// TIA Portal project "PID_1" (V16)

(* hardware
DEVICE "S71500/ET200MP station_1"  S7-1500 station
   slot 0: "Rail_0"  Rack  6ES7 590-1***0-0AA0
   slot 1: "PLC_1"  CPU 1511C-1 PN  6ES7 511-1CK01-0AB0  V2.8
      slot 3: "CPU display_1"  6ES7591-1AA00-0AA0
      slot 32768: "PROFINET interface_1"  X1
         slot 32769: "Port_1"  X1 P1
         slot 32770: "Port_2"  X1 P2
      slot 34817: "Virtual CP interface port_1"  Virtual CP interface port  Virtual CP interface port
DEVICE "HMI_1"  KTP700 Basic PN
   slot 0: "HMI_1"  KTP700 Basic PN  6AV2 123-2GB03-0AX0  16.0.0.0
   slot 1: "HMI_RT_1"  KTP700 Basic PN  6AV2 123-2GB03-0AX0  16.0.0.0
   slot 5: "HMI_1.IE_CP_1"  PROFINET Interface  16.0.0.0
      slot 1: "PROFINET Interface_1"  PROFINET Interface
         slot 1: "Port_1"  Port
*)

// ===== PLC "PLC_1"  CPU 1511C-1 PN =====

VAR_GLOBAL   // PLC tag table "Default tag table"
   "Fill level Tank" AT %IW0 : Int;
   "Analog Output" AT %QW0 : Int;
   "Empty Tank" AT %I0.0 : Bool;
   "Fill In Tank" AT %I0.1 : Bool;
   "LED Indicator" AT %Q4.0 : Bool;
END_VAR

VAR_GLOBAL   // PLC tag table "Outputs"
   "Solenoid_on/off" AT %Q0.0 : Bool;
   "Heater_on/off" AT %Q0.1 : Bool;
   "Relay KF1_Pump mode" AT %Q0.2 : Bool;
   "Pump_on/off" AT %Q0.3 : Bool;
   "KF6_Proportional valve" AT %Q0.4 : Bool;
   "KF2_Fan" AT %Q0.5 : Bool;
   "Pump_P101" AT %QW96 : Int;
END_VAR

VAR_GLOBAL   // PLC tag table "Inputs"
   "Flow_Rate_Sensor" AT %I0.0 : Bool;
   "Float_switch_overflow" AT %I0.1 : Bool;   // S111
   "Float_switch_threshold" AT %I0.2 : Bool;   // S112
   "Low_Level_Capacitive_Sensor" AT %I0.3 : Bool;   // B114
   "High_Level_Capacitive_Sensor" AT %I0.4 : Bool;   // B113
   "Micro_switch_valve_closed" AT %I0.5 : Bool;
   "Micro_switch_valve_open" AT %I0.6 : Bool;
   "Ultrasonic_Sensor" AT %IW96 : Int;
END_VAR

VAR_GLOBAL   // PLC tag table "Factory tags"
   "FactoryIO_running" AT %I0.7 : Bool;
   "Ultrasonic_Sensor_factory" AT %ID30 : Real;
   "Fill valve" AT %QD30 : Real;
   "Discharge valve" AT %QD34 : Real;
   "SP" AT %QD38 : DInt;
   "Flow meter" AT %ID34 : Real;
   "setpoint" AT %ID38 : DInt;
   "PV" AT %QD42 : Real;
END_VAR

// folder: Sys_par

DATA_BLOCK "parameters"   // DB4
{ S7_Optimized_Access := 'TRUE' }
VERSION : 0.1
   VAR
      "Process Value" : Real;
      setpoint : Int := 0;
      flowrate : Real;
      ModeActivate : Bool;
      ManualEnable : Bool;
      ManualValue : Real := 80.0;
      Mode : Int;
      Reset : Bool;
   END_VAR
BEGIN
END_DATA_BLOCK

// folder: (top level)

FUNCTION "height_conversion" : Void   // FC3, LAD
{ S7_Optimized_Access := 'TRUE' }
VERSION : 0.1
   VAR_INPUT
      height_sensor : Real;
      height_setpoint : Int;
   END_VAR
   VAR_OUTPUT
      scaled_height : Real;
      scaled_setpoint : Real;
   END_VAR
   VAR_TEMP
      norm_height : Real;
      norm_setpoint : Real;
   END_VAR
BEGIN

REGION Network 1: Height Conversion
   // 1. Normalize the sensor output data between 0.0 and 1.0
   // 2. Scale the normalized data between minimum and maximum scale reading
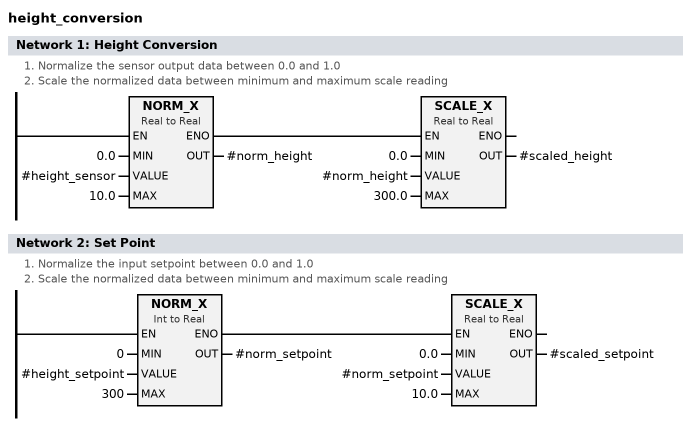
   RUNG wire#powerrail
      { S7_Templates := "[SrcType := Real, DestType := Real]" } Normalize(min := 0.0, value := #height_sensor, max := 10.0, out => #norm_height)
      { S7_Templates := "[SrcType := Real, DestType := Real]" } Scale(min := 0.0, value := #norm_height, max := 300.0, out => #scaled_height)
   END_RUNG
   // the same network as SCL:
   #norm_height := NORM_X(MIN := 0.0, VALUE := #height_sensor, MAX := 10.0);
   #scaled_height := SCALE_X(MIN := 0.0, VALUE := #norm_height, MAX := 300.0);
END_REGION

REGION Network 2: Set Point
   // 1. Normalize the input setpoint between 0.0 and 1.0
   // 2. Scale the normalized data between minimum and maximum scale reading
   RUNG wire#powerrail
      { S7_Templates := "[SrcType := Int, DestType := Real]" } Normalize(min := 0, value := #height_setpoint, max := 300, out => #norm_setpoint)
      { S7_Templates := "[SrcType := Real, DestType := Real]" } Scale(min := 0.0, value := #norm_setpoint, max := 10.0, out => #scaled_setpoint)
   END_RUNG
   // the same network as SCL:
   #norm_setpoint := NORM_X(MIN := 0, VALUE := #height_setpoint, MAX := 300);
   #scaled_setpoint := SCALE_X(MIN := 0.0, VALUE := #norm_setpoint, MAX := 10.0);
END_REGION
END_FUNCTION

FUNCTION "MHJ-PLC-Lab-Function-S71500" : Void   // FC9000, SCL
{ S7_Optimized_Access := 'TRUE' }
VERSION : 0.1
   VAR_TEMP
      Value : Byte;
      ForCounter : Int;
   END_VAR
   VAR CONSTANT
      Value_01_DW : DWord := 16#1223_5486;
      Value_02_DW : DWord := 16#A6C9_D1F5;
   END_VAR
BEGIN

   #Value:=PEEK(area := 16#82,
        dbNumber := 0,
        byteOffset := 511);
   #Value := #Value + 1;

   POKE(area := 16#82,
        dbNumber := 0,
        byteOffset := 511,
        value := #Value);

   POKE(area := 16#82,
        dbNumber := 0,
        byteOffset := 1016,
        value := #Value_01_DW);
   POKE(area := 16#82,
        dbNumber := 0,
        byteOffset := 1020,
        value := #Value_02_DW);

   FOR #ForCounter := 0 TO 63 DO
       #Value:=PEEK(area := 16#1,
            dbNumber := 0,
            byteOffset := #ForCounter);
       POKE(area := 16#81,
            dbNumber := 0,
            byteOffset := #ForCounter,
            value := #Value);
   END_FOR;
   #Value := PEEK(area := 16#1,
                  dbNumber := 0,
                  byteOffset := 512);
   POKE(area := 16#82,
        dbNumber := 0,
        byteOffset := 512,
        value := #Value);
END_FUNCTION

ORGANIZATION_BLOCK "Main"   // OB1, LAD, ProgramCycle
TITLE = "Main Program Sweep (Cycle)"
{ S7_Optimized_Access := 'TRUE' }
VERSION : 0.1
   VAR_INPUT
      Initial_Call : Bool;   // Initial call of this OB
      Remanence : Bool;   // =True, if remanent data are available
   END_VAR
BEGIN

REGION Network 1: Konnektierungsbaustein für PLC-Lab / Factory IO Function
   // Im Netzwerk 1 wird der Konnektierungsbaustein für PLC-Lab aufgerufen.
   // Dieser Aufruf darf nicht entfernt werden!
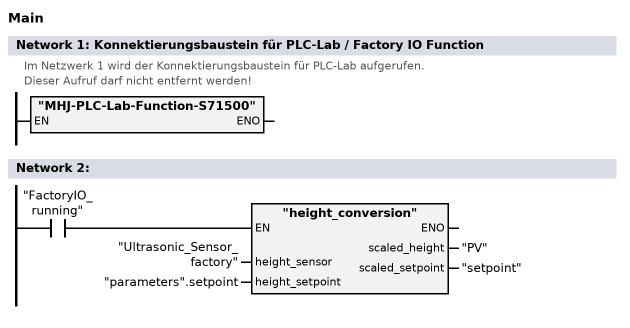
   RUNG wire#powerrail
      "MHJ-PLC-Lab-Function-S71500"()
   END_RUNG
   // the same network as SCL:
   "MHJ-PLC-Lab-Function-S71500"();
END_REGION

REGION Network 2
   RUNG wire#powerrail
      Contact( "FactoryIO_running" )
      "height_conversion"(height_sensor := "Ultrasonic_Sensor_factory", height_setpoint := "parameters".setpoint, scaled_height => "PV", scaled_setpoint => "setpoint")
   END_RUNG
   // the same network as SCL:
   IF "FactoryIO_running" THEN
       "height_conversion"(height_sensor := "Ultrasonic_Sensor_factory",
                           height_setpoint := "parameters".setpoint,
                           scaled_height => "PV",
                           scaled_setpoint => "setpoint");
   END_IF;
END_REGION
END_ORGANIZATION_BLOCK

ORGANIZATION_BLOCK "Cyclic interrupt PID"   // OB30, LAD, CyclicInterrupt
{ S7_Optimized_Access := 'TRUE' }
VERSION : 0.1
   VAR_INPUT
      Initial_Call : Bool;   // Initial call of this OB
      Event_Count : Int;   // Events discarded
   END_VAR
BEGIN

REGION Network 1
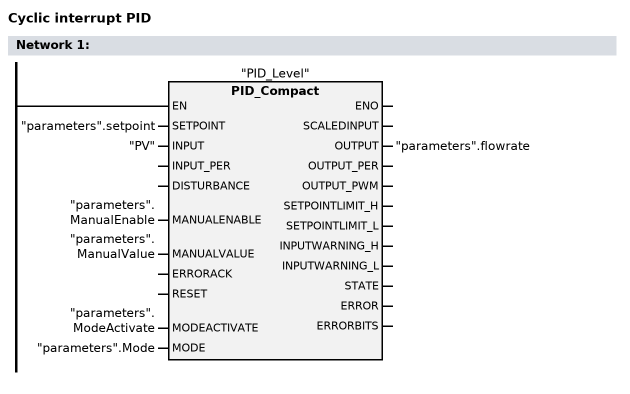
   "PID_Level"(Setpoint := "parameters".setpoint,   // PID_Compact
               Input := "PV",
               ManualEnable := "parameters".ManualEnable,
               ManualValue := "parameters".ManualValue,
               ModeActivate := "parameters".ModeActivate,
               Mode := "parameters".Mode,
               Output => "parameters".flowrate);
END_REGION
END_ORGANIZATION_BLOCK

(* ===== HMI "HMI_RT_1" =====
system functions are stored by id; their names below are inferred from use
connection "HMI_Connection_1": ETHERNET, SMART_S7_1200_OMS

HMI tags "Default tag table"
   "Tag_ScreenNumber" : UInt, internal
   "Float_switch_threshold" : Bool = PLC Float_switch_threshold AT %I0.2, 1 s
   "High_Level_Capacitive_Sensor" : Bool = PLC High_Level_Capacitive_Sensor AT %I0.4, 1 s
   "Low_Level_Capacitive_Sensor" : Bool = PLC Low_Level_Capacitive_Sensor AT %I0.3, 1 s
   "Float_switch_overflow" : Bool = PLC Float_switch_overflow AT %I0.1, 1 s
   "Micro_switch_valve_open" : Bool = PLC Micro_switch_valve_open AT %I0.6, 1 s
   "Micro_switch_valve_closed" : Bool = PLC Micro_switch_valve_closed AT %I0.5, 1 s
   "Relay KF1_Pump mode" : Bool = PLC "Relay KF1_Pump mode" AT %Q0.2, 1 s
   "KF6_Proportional valve" : Bool = PLC "KF6_Proportional valve" AT %Q0.4, 1 s
   "PV" : Real = PLC PV AT %QD42, 1 s
   "setpoint" : DInt = PLC setpoint AT %ID38, 1 s
   "PID_Compact_Level_CtrlParamsBackUp_Gain" : Real = PLC PID_Compact_Level.CtrlParamsBackUp.Gain, 1 s
   "PID_Compact_Level_CtrlParamsBackUp_Ti" : Real = PLC PID_Compact_Level.CtrlParamsBackUp.Ti, 1 s
   "PID_Compact_Level_CtrlParamsBackUp_Td" : Real = PLC PID_Compact_Level.CtrlParamsBackUp.Td, 1 s

HMI tags "Local Template"
   "_iScreenNumber" : Int, internal
   "_xState_Btn_Overview" : Bool, internal
   "_xState_Btn_Alarm" : Bool, internal
   "_xState_Btn_Recipe" : Bool, internal
   "_xState_Btn_Settings" : Bool, internal
   "_xState_Btn_Level_Overview" : Bool, internal
   "_xState_Btn_Level_Config" : Bool, internal
   "_xState_Btn_Alarm_Buffer" : Bool, internal

discrete alarms
   1: 'REFILL PROCESS 1 - PUMP- MOTOR CIRCUT BREAKER', class Errors
   2: 'REFILL PROCESS 1 - PUMP- LOCAL ISOLATOR FAULT', class Errors bit 0
   3: 'REFILL PROCESS 1 - PUMP- RUNNING FEEDBACK FAULT', class Errors bit 0
   4: 'REFILL PROCESS 1 - VALVE-NOT OPENING', class Errors bit 0
   5: 'SUPPLY-TANK-LOW LEVEL FAULT', class Errors bit 0
   6: 'SUPPLY-TANK-NOT OPENING FAULT', class Errors bit 0
   7: 'SUPPLY-TANK-HIGH LEVEL WARNING', class Warnings bit 0
   8: 'PROCESS-TANK-HIGH LEVEL ERROR', class Errors bit 0

graphic list "Graphic_Alarm_Reset": 0 'Graphic_49'; 1 'Graphic_50'

graphic list "Graphic_Return_Previous_Screen": 0..1 'Graphic_52'

graphic list "Graphic_Buffer_Screen": 0..1 'Graphic_54'

graphic list "GraphList_Btn_Template_Overview": 0 'Graphic_19'; 1 'Graphic_18'

graphic list "GraphList_Btn_Template_Alarm": 0 'Graphic_16'; 1 'Graphic_17'

graphic list "GraphList_Btn_Template_Recipe": 0 'Graphic_14'; 1 'Graphic_15'

graphic list "GraphList_Btn_Template_Settings": 0 'Graphic_13'; 1 'Graphic_12'

graphic list "GraphList_Pump": 0 'Graphic_27'; 1 'Graphic_26'

graphic list "GraphList_Proportional_Valve": 0 'Graphic_45'; 1 'Graphic_46'

screen "Overview" 800x480, template "Template"
   on GenerateScreen: SetBit("_xState_Btn_Overview")
   on ClearScreen: ResetBit("_xState_Btn_Overview")
   Button "Button_1" at 140,201 size 182x58; TextOff 'Level Control'; PictureOff "level_ind"
      on Release: ActivateScreen("Level OverView", 0)
   Button "Button_2" at 377,203 size 183x54; TextOff 'Flow Control'; PictureOff "level_ind"
   Button "Button_3" at 143,284 size 182x58; TextOff 'Level Control'; PictureOff "level_ind"
      on Release: ActivateScreen("Level OverView", 0)
   Button "Button_4" at 377,283 size 182x58; TextOff 'Level Control'; PictureOff "level_ind"
      on Release: ActivateScreen("Level OverView", 0)

screen "Recipe" 800x480, template "Template"
   on GenerateScreen: SetBit("_xState_Btn_Recipe")
   on ClearScreen: ResetBit("_xState_Btn_Recipe")

screen "Alarm" 800x480, template "Template"
   on GenerateScreen: SetBit("_xState_Btn_Alarm")
   on ClearScreen: ResetBit("_xState_Btn_Alarm")
   AlarmView "Alarm view_1" at 5,48 size 592x422
   Button "Template_Button_4" at 600,409 size 83x58; TextOff 'Text'; PictureList "GraphList_Btn_Template_Settings"; PictureOff "Graphic_49"; PictureOn "Graphic_50"
      ProcessValue <- "_xState_Btn_Settings"
   Button "Template_Button_1" at 600,48 size 83x58; TextOff 'Text'; PictureList "GraphList_Btn_Template_Settings"; PictureOff "Graphic_54"; PictureOn "Graphic_50"
      on Release: ActivateScreen("Alarm Buffer", 0)
      ProcessValue <- "_xState_Btn_Settings"

screen "Settings" 800x480, template "Template"
   on GenerateScreen: SetBit("_xState_Btn_Settings")
   on ClearScreen: ResetBit("_xState_Btn_Settings")

screen "Level OverView" 800x480, template "Template"
   on GenerateScreen: SetBit("_xState_Btn_Level_Overview")
   on ClearScreen: ResetBit("_xState_Btn_Level_Overview")
   GraphicView "Graphic view_4" at 128,89 size 150x187; Picture "Graphic_25"
   GraphicView "Graphic view_1" at 416,163 size 148x178; Picture "Graphic_25"
   Circle "Circle_4" at 107,186 size 25x25
      Appearance <- "Float_switch_threshold"
   Circle "Circle_2" at 477,138 size 25x25
      Appearance <- "Float_switch_overflow"
   Circle "Circle_3" at 392,185 size 25x25
      Appearance <- "High_Level_Capacitive_Sensor"
   Circle "Circle_1" at 565,285 size 25x25
      Appearance <- "Low_Level_Capacitive_Sensor"
   GraphicView "Graphic view_21" at 319,78 size 45x23; Picture "Graphic_40"
   GraphicView "Graphic view_25" at 222,281 size 40x21; Picture "Graphic_40"
   GraphicView "Graphic view_18" at 85,270 size 31x44; Picture "Graphic_39"
   GraphicView "Graphic view_20" at 502,367 size 51x31; Picture "Graphic_40"
   Line "Line_8" at 130,197 size 140x1
      Appearance <- "Float_switch_threshold"
   Bar "Bar_1" at 140,124 size 128x115; MinimumValue 0; MaximumValue 10
      ProcessValue <- "PV"
   Button "Button_1" at 432,372 size 43x52; TextOff 'Text'; PictureList "GraphList_Pump"
      ProcessValue <- "Relay KF1_Pump mode"
   GraphicView "Graphic view_2" at 116,382 size 322x34; Picture "Graphic_28"
   GraphicView "Graphic view_7" at 81,383 size 36x32; Picture "Graphic_32"
   GraphicView "Graphic view_3" at 83,310 size 34x75; Picture "Graphic_33"
   GraphicView "Graphic view_5" at 111,211 size 30x34; Picture "Graphic_28"
   GraphicView "Graphic view_6" at 474,333 size 34x38; Picture "Graphic_33"
   GraphicView "Graphic view_8" at 474,363 size 35x41; Picture "Graphic_36"
   GraphicView "Graphic view_9" at 191,258 size 34x22; Picture "Graphic_33"
   GraphicView "Graphic view_10" at 259,275 size 173x34; Picture "Graphic_28"
   GraphicView "Graphic view_11" at 266,116 size 27x34; Picture "Graphic_28"
   GraphicView "Graphic view_12" at 357,71 size 137x34; Picture "Graphic_28"
   GraphicView "Graphic view_13" at 524,71 size 83x34; Picture "Graphic_28"
   GraphicView "Graphic view_14" at 547,187 size 59x34; Picture "Graphic_28"
   GraphicView "Graphic view_15" at 604,98 size 34x94; Picture "Graphic_33"
   GraphicView "Graphic view_16" at 194,60 size 31x41; Picture "Graphic_37"
   GraphicView "Graphic view_17" at 190,276 size 36x32; Picture "Graphic_32"
   Line "Line_6" at 446,87 size 46x0
      Visibility <- "Micro_switch_valve_closed"
   Line "Line_7" at 529,88 size 42x0
      Visibility <- "Micro_switch_valve_open"
   GraphicView "Graphic view_19" at 290,114 size 37x37; Picture "Graphic_42"
   GraphicView "Graphic view_23" at 291,104 size 34x16; Picture "Graphic_33"
   GraphicView "Graphic view_24" at 292,75 size 33x31; Picture "Graphic_43"
   GraphicView "Graphic view_26" at 84,212 size 33x33; Picture "Graphic_43"
   GraphicView "Graphic view_27" at 83,241 size 34x38; Picture "Graphic_33"
   GraphicView "Graphic view_28" at 544,366 size 30x34; Picture "Graphic_28"
   GraphicView "Graphic view_29" at 603,186 size 37x37; Picture "Graphic_42"
   GraphicView "Graphic view_30" at 603,70 size 37x37; Picture "Graphic_44"
   Button "Button_2" at 491,67 size 36x41; TextOff 'Text'; PictureList "GraphList_Proportional_Valve"
      ProcessValue <- "KF6_Proportional valve"
   GraphicView "Graphic view_31" at 560,343 size 82x83; Picture "Graphic_48"
   Button "Button_3" at 1,0 size 157x40; TextOff 'OverView'
      Appearance <- "_xState_Btn_Level_Overview"
   Button "Button_4" at 162,0 size 157x40; TextOff 'Configuration'
      on Release: ActivateScreen("Level Config", 0)
      Appearance <- "_xState_Btn_Level_Config"
   TextField "Text field_1" at 70,162 size 45x23; Text 'S112'
   TextField "Text field_2" at 224,50 size 46x23; Text 'B102'
   TextField "Text field_3" at 340,186 size 46x23; Text 'B113'
   TextField "Text field_4" at 594,287 size 46x23; Text 'B114'
   TextField "Text field_5" at 424,140 size 45x23; Text 'S111'
   TextField "Text field_6" at 466,48 size 113x20; Text 'Proportion valve'
   TextField "Text field_7" at 115,286 size 46x23; Text 'V101'
   TextField "Text field_8" at 221,302 size 46x23; Text 'V110'
   TextField "Text field_9" at 504,396 size 46x23; Text 'V105'
   TextField "Text field_10" at 319,103 size 46x23; Text 'V112'
   TextField "Text field_11" at 508,138 size 82x20; Text 'Float switch'
   TextField "Text field_12" at 580,266 size 101x20; Text 'Low Level Cap.'
   TextField "Text field_13" at 288,165 size 103x20; Text 'High Level Cap.'
   TextField "Text field_14" at 56,141 size 82x20; Text 'Float switch'
   TextField "Text field_15" at 224,68 size 69x20; Text 'Ultrasonic'
   TextField "Text field_16" at 429,353 size 40x20; Text 'Pump'

screen "Level Config" 800x480, template "Template"
   on GenerateScreen: SetBit("_xState_Btn_Level_Config")
   on ClearScreen: ResetBit("_xState_Btn_Level_Config")
   TrendView "Trend view_1" at 38,167 size 644x300
   IOField "I/O field_1" at 442,76 size 105x27; FormatPattern 999.99
      ProcessValue <- "PID_Compact_Level_CtrlParamsBackUp_Gain"
   IOField "I/O field_2" at 442,105 size 105x27; FormatPattern 99.99
      ProcessValue <- "PID_Compact_Level_CtrlParamsBackUp_Ti"
   IOField "I/O field_3" at 442,135 size 105x27; FormatPattern 99.99
      ProcessValue <- "PID_Compact_Level_CtrlParamsBackUp_Td"
   TextField "Text field_1" at 553,80 size 107x23; Text 'Proportional'
   TextField "Text field_2" at 552,108 size 71x23; Text 'Integral'
   TextField "Text field_3" at 552,136 size 89x23; Text 'Derivative'
   Button "Button_1" at 442,47 size 218x28; TextOff 'Save PID Parameters'
   Button "Button_2" at 299,59 size 96x45; TextOff 'Enable'
   Button "Button_5" at 299,116 size 96x41; TextOff 'Disable'
   IOField "I/O field_4" at 32,69 size 105x33; FormatPattern s999999999.999
      ProcessValue <- "setpoint"
   TextField "Text field_4" at 148,76 size 75x23; Text 'SetPoint'
   IOField "I/O field_5" at 33,112 size 105x33
      ProcessValue <- "PV"
   TextField "Text field_5" at 145,118 size 118x23; Text 'Process Value'
   Button "Button_3" at 1,0 size 157x40; TextOff 'OverView'
      on Release: ActivateScreen("Level OverView", 0)
      Appearance <- "_xState_Btn_Level_Overview"
   Button "Button_4" at 162,0 size 157x40; TextOff 'Configuration'
      on Release: ActivateScreen("Level Config", 0)
      Appearance <- "_xState_Btn_Level_Config"

screen "Alarm Buffer" 800x480, template "Template"
   on GenerateScreen: SetBit("_xState_Btn_Alarm_Buffer")
   on ClearScreen: ResetBit("_xState_Btn_Alarm_Buffer")
   AlarmView "Alarm view_1" at 5,48 size 592x422
   Button "Template_Button_4" at 600,49 size 83x58; TextOff 'Text'; PictureList "GraphList_Btn_Template_Settings"; PictureOff "Graphic_52"; PictureOn "Graphic_50"
      on Release: function_efd93a16()
      ProcessValue <- "_xState_Btn_Settings"

Template "Template" 800x480
   Button "Template_Button_1" at 694,1 size 100x75; TextOff 'Text'; PictureList "GraphList_Btn_Template_Overview"
      on Release: ActivateScreen("Overview", 0)
      ProcessValue <- "_xState_Btn_Overview"
   Button "Template_Button_2" at 694,79 size 100x75; TextOff 'Text'; PictureList "GraphList_Btn_Template_Alarm"
      on Release: ActivateScreen("Alarm", 0)
      ProcessValue <- "_xState_Btn_Alarm"
   Button "Template_Button_3" at 694,157 size 100x75; TextOff 'Text'; PictureList "GraphList_Btn_Template_Recipe"
      on Release: ActivateScreen("Recipe", 0)
      ProcessValue <- "_xState_Btn_Recipe"
   Button "Template_Button_4" at 693,235 size 100x75; TextOff 'Text'; PictureList "GraphList_Btn_Template_Settings"
      on Release: ActivateScreen("Settings", 0)
      ProcessValue <- "_xState_Btn_Settings"
   TextField "Template_Text field_3" at 692,351 size 90x23; Text 'Start/stop'
*)